# EPICS substitutions: ThingyApp/Db/nodes.substitutions
file "nodes.template" {

# MAX_NODES is defined in ThingyApp/src/thingyAggregator.h and must match SERVER_COUNT defined
# in the Thingy firmware.

# NodeID can not exceed (MAX_NODES - 1) for nodes

pattern { Sys,	Dev,				NodeID}

{ "XF:10IDB",	"{THINGY:001}",		0}
{ "XF:10IDB",	"{THINGY:002}",		1}
{ "XF:10IDB",	"{THINGY:003}",		2}
{ "XF:10IDB",	"{THINGY:004}",		3}

}
